{attribute 'qualified_only'}
VAR_GLOBAL
    fbDiagnosticMessageDiagnosticCodeParser_Test_WhenEmergencyErrorCodeExpectEmergencyErrorCode : ULINT;
    fbDiagnosticMessageDiagnosticCodeParser_Test_WhenManufacturerSpecificExpectManufacturerSpecific : ULINT;
    fbDiagnosticMessageDiagnosticCodeParser_Test_WhenProfileSpecificExpectProfileSpecific : ULINT;
    fbDiagnosticMessageDiagnosticCodeParser_Test_WhenReservedForFutureUseExpectReservedForFutureUse : ULINT;

    fbDiagnosticMessageFlagsParser_Test_WhenInfoMessageExpectInfoMessageGlobalTimestampAndZeroParameters : ULINT;
    fbDiagnosticMessageFlagsParser_Test_WhenWarningMessageExpectWarningMessageLocalTimestampAndTwoParameters : ULINT;
    fbDiagnosticMessageFlagsParser_Test_WhenErrorMessageExpectErrorMessageLocalTimestampAndFourParameters : ULINT;
    fbDiagnosticMessageFlagsParser_Test_WhenReservedForFutureUseMessageExpectReservedForFutureUseMessageLocalTimestampAnd33Parameters : ULINT;    

    fbDiagnosticMessageParser_Test_TestWithEmergencyMessage : ULINT;
    fbDiagnosticMessageParser_Test_TestWithManufacturerSpecificMessage : ULINT;
    fbDiagnosticMessageParser_Test_TestWithUnspecifiedMessageMessage : ULINT;
    fbDiagnosticMessageParser_Test_TestWithUnspecifiedMessageMessage_ParameterVariant : ULINT;

    fbDiagnosticMessageTextIdentityParser_Test_WhenTextIdentityLowExpectTextIdentity0 : ULINT;
    fbDiagnosticMessageTextIdentityParser_Test_WhenTextIdentityHighExpectTextIdentity65535 : ULINT;
    fbDiagnosticMessageTextIdentityParser_Test_WhenTextIdentityMedExpectTextIdentity34500 : ULINT;

    fbDiagnosticMessageTimeStampParser_Test_TestWithTimestampZeroTimeExpectCurrentTime : ULINT;
    fbDiagnosticMessageTimeStampParser_Test_TestWithValidTimestampExpectSameTimestamp : ULINT;
END_VAR

(* stored: Version 1.1.0.1, ProductVersion 3.1.4022.18
   GVL GVL: Id {2ee23b30-e6fe-4c1b-b0ea-d35d6a0d8c22} *)
